Staubli VAL3: setAllSpeed.pgx

program setAllSpeed(num x_nNewValue, num x_nOldValue)
  local num i
  local num l_nSize
begin
end
